INTERFACE I_Payload EXTENDS __System.IQueryInterface

END_INTERFACE

(* stored: Version 1.1.0.1, ProductVersion 3.1.4024.2
   Itf I_Payload: Id {857351d2-fe84-439c-8980-f8e376bc611d} *)
